// LS Electric XG5000 project: IP_STC_TEST(IMAMV2)
// PLC NewPLC

PROGRAM NewProgram (task: Scan Program)

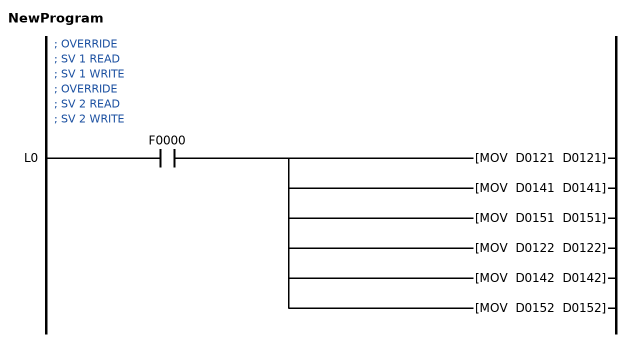
; L0
LOAD      F0000
MOV       D0121 D0121
MOV       D0141 D0141
MOV       D0151 D0151
MOV       D0122 D0122
MOV       D0142 D0142
MOV       D0152 D0152
// output comment: OVERRIDE
// output comment: SV 1 READ
// output comment: SV 1 WRITE
// output comment: OVERRIDE
// output comment: SV 2 READ
// output comment: SV 2 WRITE